(* Logix 5000 project; controller NorthLineDepalletizerPLC vendor 1 type 14 code 106 rev 33.11; software revision 33.00; part 3 of 4 *)
(* tags used below, declared in another part *)
   AcknowledgeHeightCheck : ALIAS FOR YRC1000_Rbt_Ctlr:O.Data[4].4;
   AcknowledgeLevelCheck : ALIAS FOR YRC1000_Rbt_Ctlr:O.Data[6].4;
   AcknowledgePalletTooTall : ALIAS FOR YRC1000_Rbt_Ctlr:O.Data[7].4;
   ActiveUserFrame : DINT;   // Currently Active Pallet
   AirPressure : ALIAS FOR YRC1000_Rbt_Ctlr:I.Data[1].4;
   Alarm : ALIAS FOR YRC1000_Rbt_Ctlr:I.Data[8].3;
   AngleHeightCheck : ALIAS FOR YRC1000_Rbt_Ctlr:I.Data[10].4;
   AtHomePosition : ALIAS FOR YRC1000_Rbt_Ctlr:I.Data[5].2;
   CameraFailed : ALIAS FOR YRC1000_Rbt_Ctlr:O.Data[5].7;
   CapacitiveSensorValue : DINT;
   CoilType : DINT;   // 1: 17" 2: 30" 3: 41"
   CompleteState : DINT;
   ConveyorApproach : YRC1000_POSITION_VAR;
   ConveyorBeforePlace : YRC1000_POSITION_VAR;
   ConveyorIn : YRC1000_POSITION_VAR;
   ConveyorOver : YRC1000_POSITION_VAR;
   Corner1Dist : DINT;
   Corner2Dist : DINT;
   Corner3Dist : DINT;
   Corner4Dist : DINT;
   Cos30 : REAL;
   Cos45 : REAL;
   CurrentPos : REAL[6];   // Current position of the active TCP on the robot
   CurrentPosition_micro : YRC1000_POSITION_VAR;
   delay_ActiveUserFrame : TIMER;
   delay_CurrentPos : TIMER;
   delay_Read_PartCount : TIMER;
   delay_Read_RobotCurrentTask : TIMER;
   DiffHeightCheckVal : DINT;   // Difference between the highest and shortest corners of a pallet
   DistanceSensorValue_micro : DINT;
   DoorRequestAccess : ALIAS FOR YRC1000_Rbt_Ctlr:I.Data[1].0;
   DoorUnlocked : ALIAS FOR YRC1000_Rbt_Ctlr:I.Data[1].7;
   err_CameraFailed : BOOL;
   err_HeightCheckInconsistent : ALIAS FOR YRC1000_Rbt_Ctlr:O.Data[6].3;
   err_RobotPickupFailed : ALIAS FOR YRC1000_Rbt_Ctlr:I.Data[10].3;
   ExternalHold : ALIAS FOR YRC1000_Rbt_Ctlr:O.Data[0].1;
   Gripper_Extended : ALIAS FOR YRC1000_Rbt_Ctlr:O.Data[5].0;
   Gripper_HoldingPart : ALIAS FOR YRC1000_Rbt_Ctlr:O.Data[4].7;
   Gripper_Retracted : ALIAS FOR YRC1000_Rbt_Ctlr:O.Data[5].1;
   HeightCheck1 : ALIAS FOR YRC1000_Rbt_Ctlr:I.Data[9].0;
   HeightCheck2 : ALIAS FOR YRC1000_Rbt_Ctlr:I.Data[9].1;
   HeightCheck3 : ALIAS FOR YRC1000_Rbt_Ctlr:I.Data[9].2;
   HeightCheck4 : ALIAS FOR YRC1000_Rbt_Ctlr:I.Data[9].3;
   HeightCheckAngled : REAL;
   HeightCheckAvg : DINT;
   HeightCheckTotal : DINT;
   HighestCorner : DINT;   // Index of the highest corner on a quad-stack pallet
   i : DINT;
   IFM_Device_Disconnected : BOOL;
   InHomePosition : ALIAS FOR YRC1000_Rbt_Ctlr:O.Data[5].6;
   InRemote : ALIAS FOR YRC1000_Rbt_Ctlr:I.Data[8].5;
   j : DINT;
   JobResults : PatternResult[4];   // Organized results from the most recent camera image
   LeftConveyorPresent : ALIAS FOR YRC1000_Rbt_Ctlr:O.Data[7].6;
   LeftEdgeFound : ALIAS FOR YRC1000_Rbt_Ctlr:O.Data[6].7;
   LeftPalletComplete : ALIAS FOR YRC1000_Rbt_Ctlr:O.Data[4].0;
   LeftPalletPresent : ALIAS FOR YRC1000_Rbt_Ctlr:O.Data[7].1;
   LevelCheck1 : ALIAS FOR YRC1000_Rbt_Ctlr:I.Data[10].7;
   LevelCheck2 : ALIAS FOR YRC1000_Rbt_Ctlr:I.Data[11].0;
   LevelCheck3 : ALIAS FOR YRC1000_Rbt_Ctlr:I.Data[11].1;
   LevelCheckBad : ALIAS FOR YRC1000_Rbt_Ctlr:O.Data[7].3;
   LevelCheckDone : ALIAS FOR YRC1000_Rbt_Ctlr:O.Data[6].5;
   LevelCheckStopPoint : DINT;
   LoopsFound : BOOL;   // Used to determine if we are looking at the wrong end of a single-stack coil
   MaxHeightCheckVal : DINT;
   MinHeightCheckVal : DINT;
   msg_Read_ActiveUserFrame : MESSAGE;
   msg_Read_CurrentPosition : MESSAGE;
   msg_Read_CurrentRobotTask : MESSAGE;
   msg_Read_PartCount : MESSAGE;
   msg_Read_SearchLocation : MESSAGE;
   msg_Write_ActiveUserFrame : MESSAGE;
   msg_Write_CoilLocation : MESSAGE;
   msg_Write_CoilType : MESSAGE;
   msg_Write_ConveyorApproach : MESSAGE;
   msg_Write_ConveyorBeforePlace : MESSAGE;
   msg_Write_ConveyorIn : MESSAGE;
   msg_Write_ConveyorOver : MESSAGE;
   msg_Write_HeightCheckAverage : MESSAGE;
   msg_Write_HighestCorner : MESSAGE;
   msg_Write_PartCount : MESSAGE;
   msg_Write_SearchLocation : MESSAGE;
   ons_IncPickFailCount : BOOL;
   ons_Reset_PC_HeightCheck : BOOL;
   ons_StartHeightCheck : BOOL;
   ons_StartLevelCheck : BOOL;
   p : DINT;
   PalletTooTall : ALIAS FOR YRC1000_Rbt_Ctlr:I.Data[9].6;
   PartCount : DINT;   // Number of coils the robot has placed on either conveyor
   PartID : DINT;
   PartLength_Current : DINT;   // 17" = 432 mm 30" = 762 mm 41" = 1041 mm
   PartRows_Current : DINT;
   PartThickness_Current : REAL;   // 2r = 34.1 - 34.8 mm 3r = 51.1 - 51.8 mm 4r = 68.2 - 68.9 mm
   PartWidth_Current : DINT;   // 14" = 356 mm 16" = 406 mm 20" = 508 mm 22" = 559 mm 24" = 610 mm 28" = 711 mm 32" = 813 mm
   PickFailCount : COUNTER;
   PickFailedThreeTimes : ALIAS FOR YRC1000_Rbt_Ctlr:O.Data[7].5;
   PickupErrorAcknowledge : ALIAS FOR YRC1000_Rbt_Ctlr:O.Data[5].5;
   QuadStack : ALIAS FOR YRC1000_Rbt_Ctlr:O.Data[4].3;
   Queue_PartCount : DINT[4];   // Queue of Part Counts to help keep track of what part info the Fanuc needs
   Queue_PartID : DINT[4];   // Queue of Part IDs to send to the Fanuc
   Queue_PartLength : DINT[4];   // Queue of Part Lengths to send to the Fanuc
   Queue_PartWidth : DINT[4];   // Queue of Part Widths to send to the Fanuc
   Read_ActiveUserFrame : BOOL;
   Read_CurrentPosition : BOOL;
   Read_CurrentRobotTask : BOOL;
   Read_PartCount : BOOL;
   Read_SearchLocation : BOOL;
   recovery_CameraFailed : BOOL;
   recovery_HeightCheckFailed : BOOL;
   recovery_PalletTooTall : BOOL;
   recovery_PickupFailed : BOOL;
   Reset : ALIAS FOR YRC1000_Rbt_Ctlr:I.Data[1].1;
   RightConveyorPresent : ALIAS FOR YRC1000_Rbt_Ctlr:O.Data[7].7;
   RightEdgeFound : ALIAS FOR YRC1000_Rbt_Ctlr:O.Data[7].0;
   RightPalletComplete : ALIAS FOR YRC1000_Rbt_Ctlr:O.Data[4].1;
   RightPalletPresent : ALIAS FOR YRC1000_Rbt_Ctlr:O.Data[7].2;
   RobotCurrentPalletComplete : ALIAS FOR YRC1000_Rbt_Ctlr:I.Data[10].6;
   RobotExternalEStop : ALIAS FOR YRC1000_Rbt_Ctlr:I.Data[4].1;
   RobotTeachPendantEStop : ALIAS FOR YRC1000_Rbt_Ctlr:I.Data[4].2;
   Running : ALIAS FOR YRC1000_Rbt_Ctlr:I.Data[8].0;
   RunPalletComplete : BOOL;
   SafetyCircuitBroken : ALIAS FOR YRC1000_Rbt_Ctlr:I.Data[4].0;
   SelectedJobID : DINT;
   SingleStack : ALIAS FOR YRC1000_Rbt_Ctlr:O.Data[4].2;
   StackLight_Blue : ALIAS FOR YRC1000_Rbt_Ctlr:O.Data[1].3;
   StackLight_Green : ALIAS FOR YRC1000_Rbt_Ctlr:O.Data[1].5;
   StackLight_Red : ALIAS FOR YRC1000_Rbt_Ctlr:O.Data[1].2;
   StackLight_White : ALIAS FOR YRC1000_Rbt_Ctlr:O.Data[1].1;
   StackLight_Yellow : ALIAS FOR YRC1000_Rbt_Ctlr:O.Data[1].4;
   state_HeightCheck : DINT;
   state_LevelCheck : DINT;
   state_PalletComplete : DINT;
   timer_HoldingPart : TIMER;
   ToPC_ActivePallet : DINT;
   ToPC_AirPressure : DINT;
   ToPC_CameraFailed : DINT;
   ToPC_CellStatus : DINT;
   ToPC_DoorStatus : DINT;
   ToPC_HeightCheckFailed : DINT;
   ToPC_InRemote : DINT;
   ToPC_LeftConveyorSensor : DINT;
   ToPC_LeftPalletStatus : DINT;
   ToPC_PalletTooTall : DINT;
   ToPC_PickupFailed : DINT;
   ToPC_RightConveyorSensor : DINT;
   ToPC_RightPalletStatus : DINT;
   ToPC_RobotAlarm : DINT;
   ToPC_RobotEStop : DINT;
   ToPC_RobotRunning : DINT;
   ToPC_RobotSafetyStop : DINT;
   ToPC_ToolStatus : DINT;
   Write_ActiveUserFrame : BOOL;
   write_ActiveUserFrame_L : BOOL;
   Write_ActiveUserFrame_R : BOOL;
   Write_CoilLocation : BOOL;
   Write_CoilType : BOOL;
   Write_ConveyorPositions : BOOL;
   Write_HeightCheckAverage : BOOL;
   write_HighestCorner : BOOL;
   Write_PartCount : BOOL;
   Write_SearchLocation : BOOL;
(* MainProgram, continued *)

ROUTINE PC_TagVariables   (* ladder *)
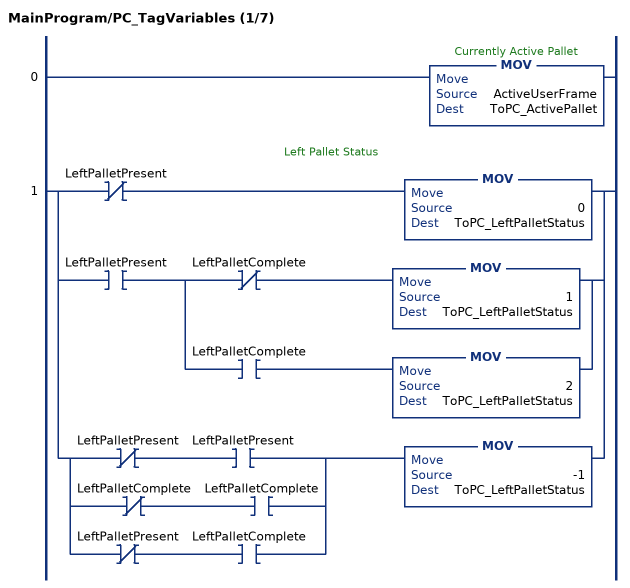
   0: MOV(ActiveUserFrame,ToPC_ActivePallet);
   // Left Pallet Status
   1: [XIO(LeftPalletPresent) MOV(0,ToPC_LeftPalletStatus) ,XIC(LeftPalletPresent) [XIO(LeftPalletComplete) MOV(1,ToPC_LeftPalletStatus) ,XIC(LeftPalletComplete) MOV(2,ToPC_LeftPalletStatus) ] ,[XIO(LeftPalletPresent) XIC(LeftPalletPresent) ,XIO(LeftPalletComplete) XIC(LeftPalletComplete) ,XIO(LeftPalletPresent) XIC(LeftPalletComplete) ] MOV(-1,ToPC_LeftPalletStatus) ];
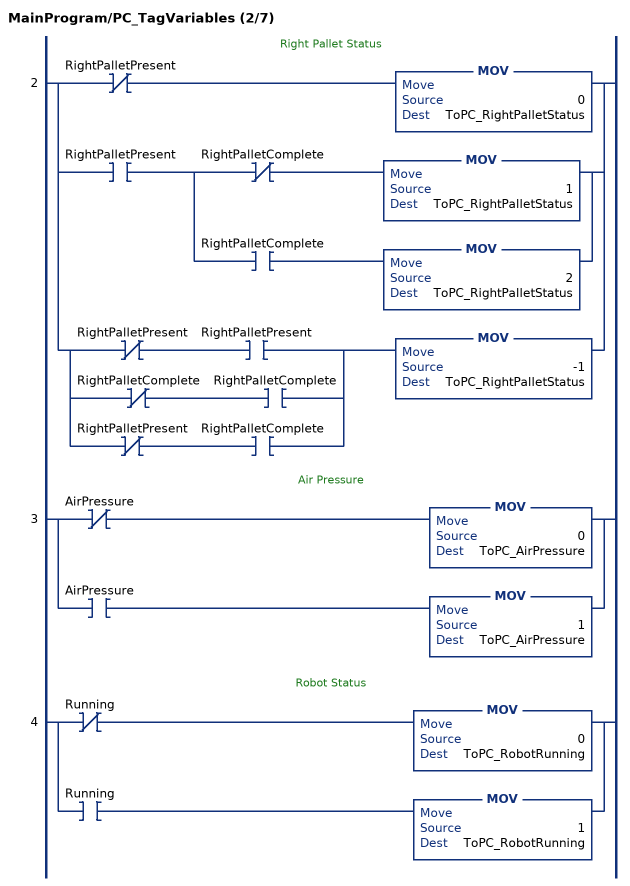
   // Right Pallet Status
   2: [XIO(RightPalletPresent) MOV(0,ToPC_RightPalletStatus) ,XIC(RightPalletPresent) [XIO(RightPalletComplete) MOV(1,ToPC_RightPalletStatus) ,XIC(RightPalletComplete) MOV(2,ToPC_RightPalletStatus) ] ,[XIO(RightPalletPresent) XIC(RightPalletPresent) ,XIO(RightPalletComplete) XIC(RightPalletComplete) ,XIO(RightPalletPresent) XIC(RightPalletComplete) ] MOV(-1,ToPC_RightPalletStatus) ];
   // Air Pressure
   3: [XIO(AirPressure) MOV(0,ToPC_AirPressure) ,XIC(AirPressure) MOV(1,ToPC_AirPressure) ];
   // Robot Status
   4: [XIO(Running) MOV(0,ToPC_RobotRunning) ,XIC(Running) MOV(1,ToPC_RobotRunning) ];
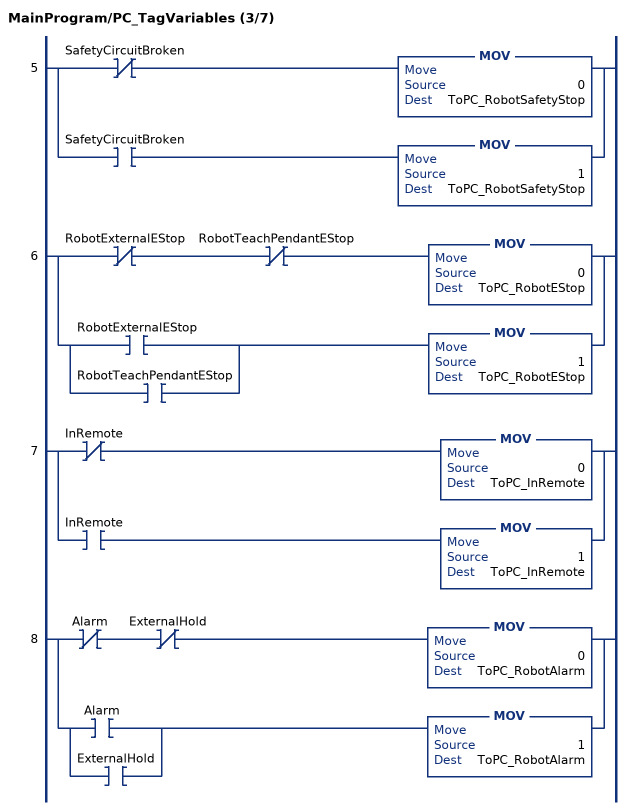
   5: [XIO(SafetyCircuitBroken) MOV(0,ToPC_RobotSafetyStop) ,XIC(SafetyCircuitBroken) MOV(1,ToPC_RobotSafetyStop) ];
   6: [XIO(RobotExternalEStop) XIO(RobotTeachPendantEStop) MOV(0,ToPC_RobotEStop) ,[XIC(RobotExternalEStop) ,XIC(RobotTeachPendantEStop) ] MOV(1,ToPC_RobotEStop) ];
   7: [XIO(InRemote) MOV(0,ToPC_InRemote) ,XIC(InRemote) MOV(1,ToPC_InRemote) ];
   8: [XIO(Alarm) XIO(ExternalHold) MOV(0,ToPC_RobotAlarm) ,[XIC(Alarm) ,XIC(ExternalHold) ] MOV(1,ToPC_RobotAlarm) ];
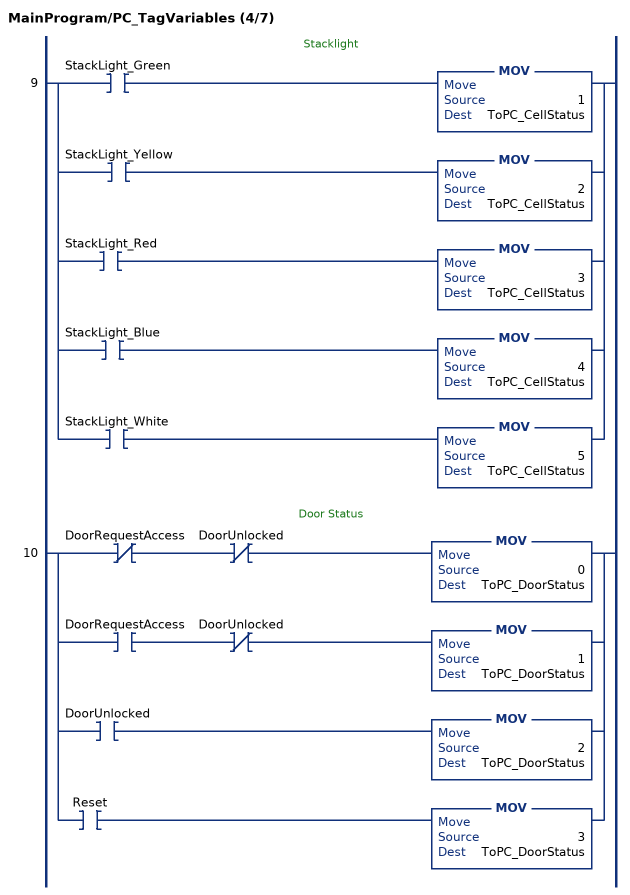
   // Stacklight
   9: [XIC(StackLight_Green) MOV(1,ToPC_CellStatus) ,XIC(StackLight_Yellow) MOV(2,ToPC_CellStatus) ,XIC(StackLight_Red) MOV(3,ToPC_CellStatus) ,XIC(StackLight_Blue) MOV(4,ToPC_CellStatus) ,XIC(StackLight_White) MOV(5,ToPC_CellStatus) ];
   // Door Status
   10: [XIO(DoorRequestAccess) XIO(DoorUnlocked) MOV(0,ToPC_DoorStatus) ,XIC(DoorRequestAccess) XIO(DoorUnlocked) MOV(1,ToPC_DoorStatus) ,XIC(DoorUnlocked) MOV(2,ToPC_DoorStatus) ,XIC(Reset) MOV(3,ToPC_DoorStatus) ];
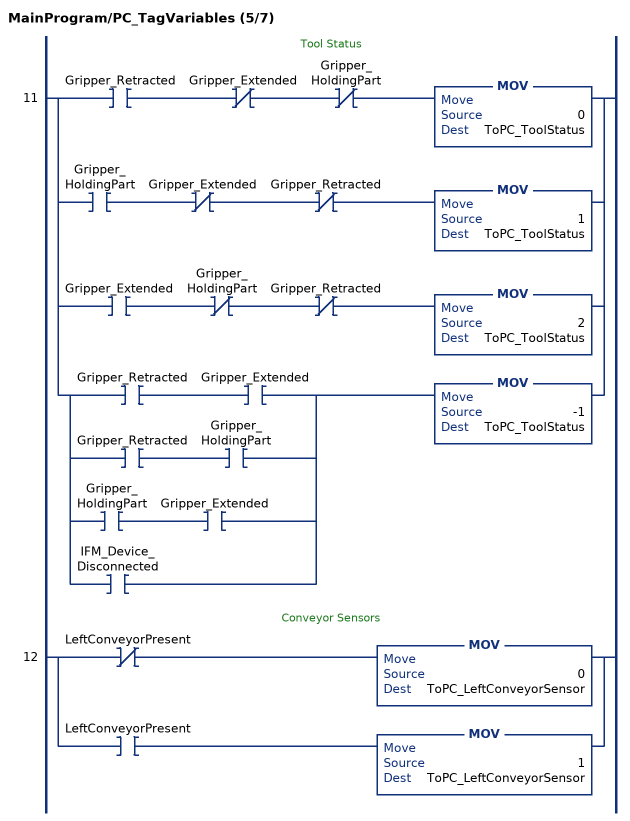
   // Tool Status
   11: [XIC(Gripper_Retracted) XIO(Gripper_Extended) XIO(Gripper_HoldingPart) MOV(0,ToPC_ToolStatus) ,XIC(Gripper_HoldingPart) XIO(Gripper_Extended) XIO(Gripper_Retracted) MOV(1,ToPC_ToolStatus) ,XIC(Gripper_Extended) XIO(Gripper_HoldingPart) XIO(Gripper_Retracted) MOV(2,ToPC_ToolStatus) ,[XIC(Gripper_Retracted) XIC(Gripper_Extended) ,XIC(Gripper_Retracted) XIC(Gripper_HoldingPart) ,XIC(Gripper_HoldingPart) XIC(Gripper_Extended) ,XIC(IFM_Device_Disconnected) ] MOV(-1,ToPC_ToolStatus) ];
   // Conveyor Sensors
   12: [XIO(LeftConveyorPresent) MOV(0,ToPC_LeftConveyorSensor) ,XIC(LeftConveyorPresent) MOV(1,ToPC_LeftConveyorSensor) ];
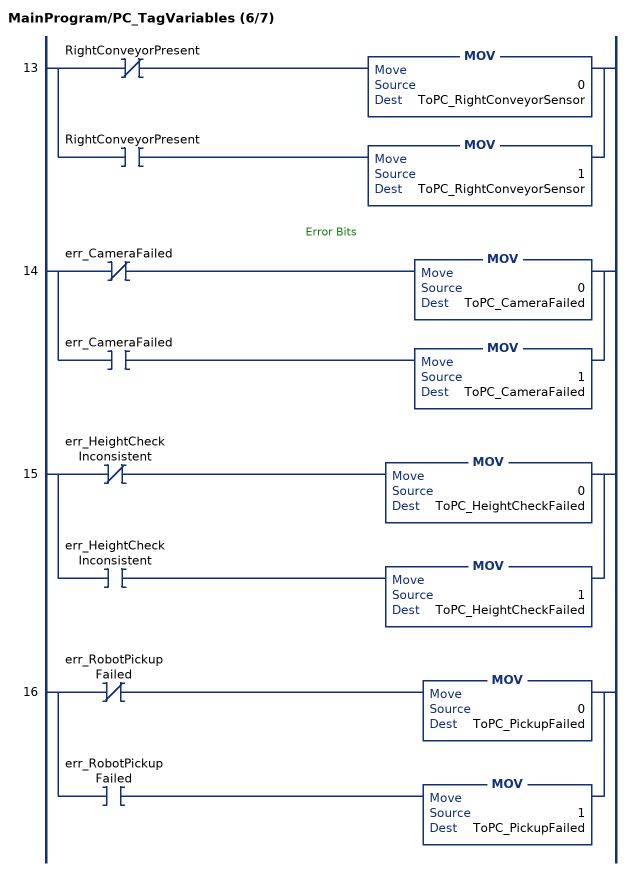
   13: [XIO(RightConveyorPresent) MOV(0,ToPC_RightConveyorSensor) ,XIC(RightConveyorPresent) MOV(1,ToPC_RightConveyorSensor) ];
   // Error Bits
   14: [XIO(err_CameraFailed) MOV(0,ToPC_CameraFailed) ,XIC(err_CameraFailed) MOV(1,ToPC_CameraFailed) ];
   15: [XIO(err_HeightCheckInconsistent) MOV(0,ToPC_HeightCheckFailed) ,XIC(err_HeightCheckInconsistent) MOV(1,ToPC_HeightCheckFailed) ];
   16: [XIO(err_RobotPickupFailed) MOV(0,ToPC_PickupFailed) ,XIC(err_RobotPickupFailed) MOV(1,ToPC_PickupFailed) ];
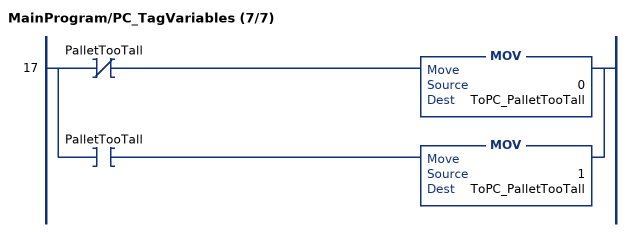
   17: [XIO(PalletTooTall) MOV(0,ToPC_PalletTooTall) ,XIC(PalletTooTall) MOV(1,ToPC_PalletTooTall) ];
END_ROUTINE

ROUTINE SaveImageResults   (* structured text *)
   /*
   	Simple loop going through all the information given by the camera after capturing an image
   	Loop through the 28 possible patterns
   	Each pattern has 4 parts: Angle, Score, X, and Y
   */
   
   for i := 0 to 2 by 1 do
   	j := i * 4;
   	JobResults[i].Angle := cam:I.InspectionResults[j];
   	JobResults[i].Score := cam:I.InspectionResults[j + 1];
   	JobResults[i].X := cam:I.InspectionResults[j + 2];
   	JobResults[i].Y := cam:I.InspectionResults[j + 3];
   end_for;
   
   if SelectedJobID = 2832 then
   	if cam:I.InspectionResults[12] > 0 then
   		LoopsFound := 1;
   	else
   		LoopsFound := 0;
   	end_if;
   end_if;
   
   if SelectedJobID = 3041 then
   	if cam:I.InspectionResults[12] > 0 then
   		LeftEdgeFound := 1;
   	else
   		LeftEdgeFound := 0;
   	end_if;
   	if cam:I.InspectionResults[13] > 0 then
   		RightEdgeFound := 1;
   	else
   		RightEdgeFound := 0;
   	end_if;
   	if cam:I.InspectionResults[14] > 0 then
   		LoopsFound := 1;
   	else
   		LoopsFound := 0;
   	end_if;
   end_if;
END_ROUTINE
END_PROGRAM

PROGRAM Motoman   (* main routine Main *)

ROUTINE AddPartToQueue   (* structured text *)
   // Determine unique Part ID that can be sent to the Fanuc
   if PartLength_Current = 432 then
   	if PartWidth_Current = 356 then
   		PartID := 1;
   	elsif PartWidth_Current = 406 then
   		PartID := 2;
   	elsif PartWidth_Current = 508 then
   		if PartRows_Current = 2 then
   			PartID := 3;
   		elsif PartRows_Current = 3 then
   			PartID := 4;
   		end_if;
   	elsif PartWidth_Current = 559 then
   		PartID := 5;
   	elsif PartWidth_Current = 610 then
   		PartID := 6;
   	elsif PartWidth_Current = 711 then
   		if PartRows_Current = 3 then
   			PartID := 7;
   		elsif PartRows_Current = 4 then
   			PartID := 8;
   		end_if;
   	elsif PartWidth_Current = 813 then
   		PartID := 9;
   	end_if;
   elsif PartLength_Current = 762 then
   	if PartRows_Current = 2 then
   		PartID := 10;
   	elsif PartRows_Current = 3 then
   		PartID := 11;
   	end_if;
   elsif PartLength_Current = 1041 then
   	if PartRows_Current = 3 then
   		PartID := 12;
   	elsif PartRows_Current = 4 then
   		PartID := 13;
   	end_if;
   end_if;
   
   // Add information about the new part to a bunch of arrays
   for p := 1 to 3 do
   	if Queue_PartID[p] = 0 then
   		Queue_PartCount[p-1] := PartCount;
   		Queue_PartID[p] := PartID;
   		Queue_PartLength[p] := PartLength_Current;
   		Queue_PartWidth[p] := PartWidth_Current;
   
   		RET();
   	end_if;
   end_for;
   
END_ROUTINE

ROUTINE CheckForHeightOutliers   (* structured text *)
   MinHeightCheckVal := 0;
   MaxHeightCheckVal := 0;
   DiffHeightCheckVal := 0;
   
   if Corner1Dist <= Corner2Dist AND Corner1Dist <= Corner3Dist AND Corner1Dist <= Corner4Dist then
   	MinHeightCheckVal := Corner1Dist;
   	HighestCorner := 1;
   elsif Corner2Dist <= Corner1Dist AND Corner2Dist <= Corner3Dist AND Corner2Dist <= Corner4Dist then
   	MinHeightCheckVal := Corner2Dist;
   	HighestCorner := 2;
   elsif Corner3Dist <= Corner1Dist AND Corner3Dist <= Corner2Dist AND Corner3Dist <= Corner4Dist then
   	MinHeightCheckVal := Corner3Dist;
   	HighestCorner := 3;
   elsif Corner4Dist <= Corner1Dist AND Corner4Dist <= Corner2Dist AND Corner4Dist <= Corner3Dist then
   	MinHeightCheckVal := Corner4Dist;
   	HighestCorner := 4;
   end_if;
   
   if Corner1Dist >= Corner2Dist AND Corner1Dist >= Corner3Dist AND Corner1Dist >= Corner4Dist then
   	MaxHeightCheckVal := Corner1Dist;
   elsif Corner2Dist >= Corner1Dist AND Corner2Dist >= Corner3Dist AND Corner2Dist >= Corner4Dist then
   	MaxHeightCheckVal := Corner2Dist;
   elsif Corner3Dist >= Corner1Dist AND Corner3Dist >= Corner2Dist AND Corner3Dist >= Corner4Dist then
   	MaxHeightCheckVal := Corner3Dist;
   elsif Corner4Dist >= Corner1Dist AND Corner4Dist >= Corner2Dist AND Corner4Dist >= Corner3Dist then
   	MaxHeightCheckVal := Corner4Dist;
   end_if;
   
   DiffHeightCheckVal := MaxHeightCheckVal - MinHeightCheckVal;
   if DiffHeightCheckVal > 25000 AND MinHeightCheckVal < 1990000 then
   	err_HeightCheckInconsistent := 1;
   else
   	err_HeightCheckInconsistent := 0;
   end_if;
END_ROUTINE

ROUTINE ConveyorVariableData   (* structured text *)
   /*
   	The only major values that change are
   		Tool_Num depending on the Part Length and
   		Axis3_Data depending on the Part Thickness
   */
   
   // Tool Number
   if PartLength_Current = 432 then
   	ConveyorApproach.Tool_Num := 8;
   	ConveyorOver.Tool_Num := 8;
   	ConveyorIn.Tool_Num := 8;
   	ConveyorBeforePlace.Tool_Num := 8;
   	ConveyorOver.Axis5_Data := 100000;
   	ConveyorIn.Axis5_Data := 100000;
   	ConveyorBeforePlace.Axis5_Data := 100000;
   elsif PartLength_Current = 762 then
   	ConveyorApproach.Tool_Num := 9;
   	ConveyorOver.Tool_Num := 9;
   	ConveyorIn.Tool_Num := 9;
   	ConveyorBeforePlace.Tool_Num := 9;
   	ConveyorOver.Axis5_Data := 100000;
   	ConveyorIn.Axis5_Data := 100000;
   	ConveyorBeforePlace.Axis5_Data :=100000;
   elsif PartLength_Current = 1041 then
   	ConveyorApproach.Tool_Num := 10;
   	ConveyorOver.Tool_Num := 10;
   	ConveyorIn.Tool_Num := 10;
   	ConveyorBeforePlace.Tool_Num := 10;
   	ConveyorOver.Axis5_Data := 80000;
   	ConveyorIn.Axis5_Data := 80000;
   	ConveyorBeforePlace.Axis5_Data := 80000;
   end_if;
   
   // Conveyor Above Z value is dependent on Part Thickness
   ConveyorApproach.Axis3_Data := (PartThickness_Current + 100) * 1000;
   ConveyorOver.Axis3_Data := (PartThickness_Current + 100) * 1000;
   ConveyorIn.Axis3_Data := (PartThickness_Current + 5) * 1000;
   ConveyorBeforePlace.Axis3_Data := (PartThickness_Current + 5) * 1000;
END_ROUTINE

ROUTINE ErrorBits   (* ladder *)
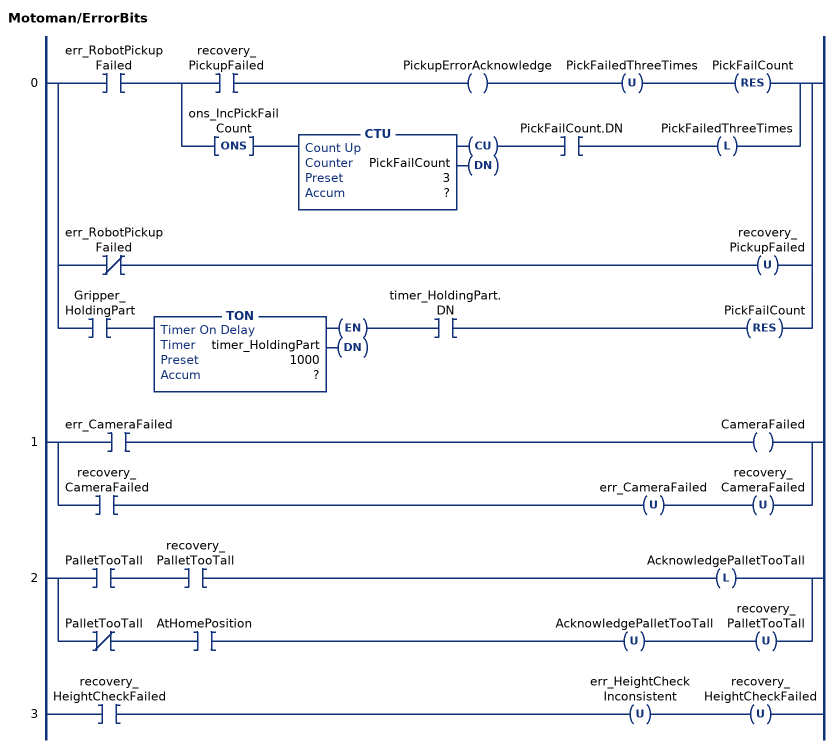
   0: [XIC(err_RobotPickupFailed) [XIC(recovery_PickupFailed) OTE(PickupErrorAcknowledge) OTU(PickFailedThreeTimes) RES(PickFailCount) ,ONS(ons_IncPickFailCount) CTU(PickFailCount,?,?) XIC(PickFailCount.DN) OTL(PickFailedThreeTimes) ] ,XIO(err_RobotPickupFailed) OTU(recovery_PickupFailed) ,XIC(Gripper_HoldingPart) TON(timer_HoldingPart,?,?) XIC(timer_HoldingPart.DN) RES(PickFailCount) ];
   1: [XIC(err_CameraFailed) OTE(CameraFailed) ,XIC(recovery_CameraFailed) OTU(err_CameraFailed) OTU(recovery_CameraFailed) ];
   2: [XIC(PalletTooTall) XIC(recovery_PalletTooTall) OTL(AcknowledgePalletTooTall) ,XIO(PalletTooTall) XIC(AtHomePosition) OTU(AcknowledgePalletTooTall) OTU(recovery_PalletTooTall) ];
   3: XIC(recovery_HeightCheckFailed)OTU(err_HeightCheckInconsistent)OTU(recovery_HeightCheckFailed);
END_ROUTINE

ROUTINE HeightCheck   (* ladder *)
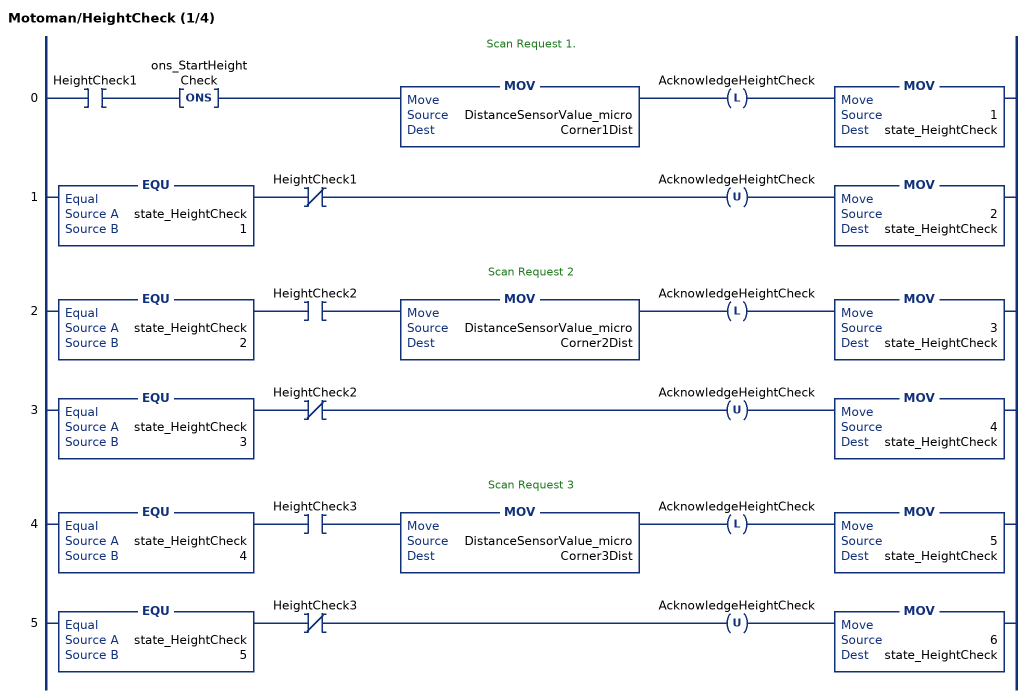
   // Scan Request 1.
   0: XIC(HeightCheck1)ONS(ons_StartHeightCheck)MOV(DistanceSensorValue_micro,Corner1Dist)OTL(AcknowledgeHeightCheck)MOV(1,state_HeightCheck);
   1: EQU(state_HeightCheck,1)XIO(HeightCheck1)OTU(AcknowledgeHeightCheck)MOV(2,state_HeightCheck);
   // Scan Request 2
   2: EQU(state_HeightCheck,2)XIC(HeightCheck2)MOV(DistanceSensorValue_micro,Corner2Dist)OTL(AcknowledgeHeightCheck)MOV(3,state_HeightCheck);
   3: EQU(state_HeightCheck,3)XIO(HeightCheck2)OTU(AcknowledgeHeightCheck)MOV(4,state_HeightCheck);
   // Scan Request 3
   4: EQU(state_HeightCheck,4)XIC(HeightCheck3)MOV(DistanceSensorValue_micro,Corner3Dist)OTL(AcknowledgeHeightCheck)MOV(5,state_HeightCheck);
   5: EQU(state_HeightCheck,5)XIO(HeightCheck3)OTU(AcknowledgeHeightCheck)MOV(6,state_HeightCheck);
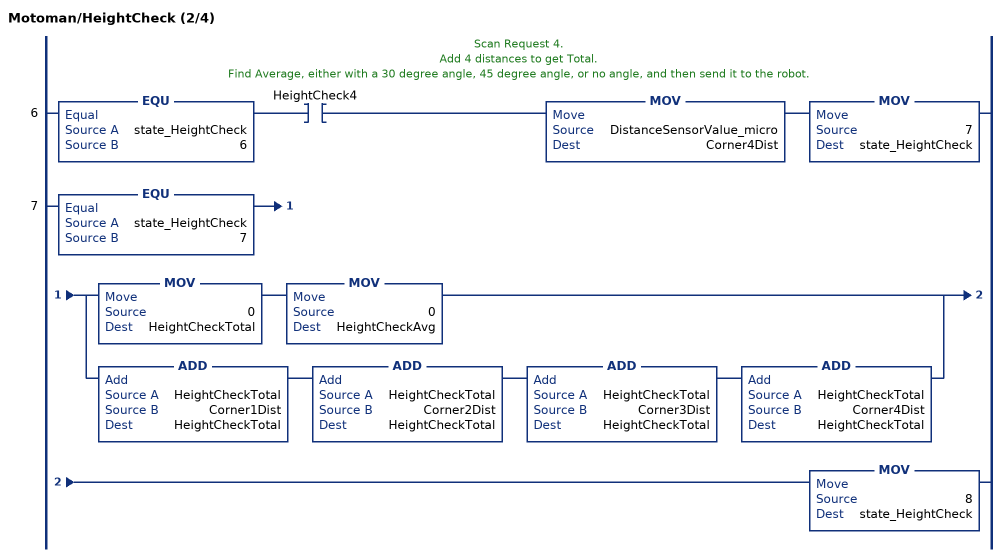
   // Scan Request 4.
   // Add 4 distances to get Total.
   // Find Average, either with a 30 degree angle, 45 degree angle, or no angle, and then send it to the robot.
   6: EQU(state_HeightCheck,6)XIC(HeightCheck4)MOV(DistanceSensorValue_micro,Corner4Dist)MOV(7,state_HeightCheck);
   7: EQU(state_HeightCheck,7)[MOV(0,HeightCheckTotal) MOV(0,HeightCheckAvg) ,ADD(HeightCheckTotal,Corner1Dist,HeightCheckTotal) ADD(HeightCheckTotal,Corner2Dist,HeightCheckTotal) ADD(HeightCheckTotal,Corner3Dist,HeightCheckTotal) ADD(HeightCheckTotal,Corner4Dist,HeightCheckTotal) ]MOV(8,state_HeightCheck);
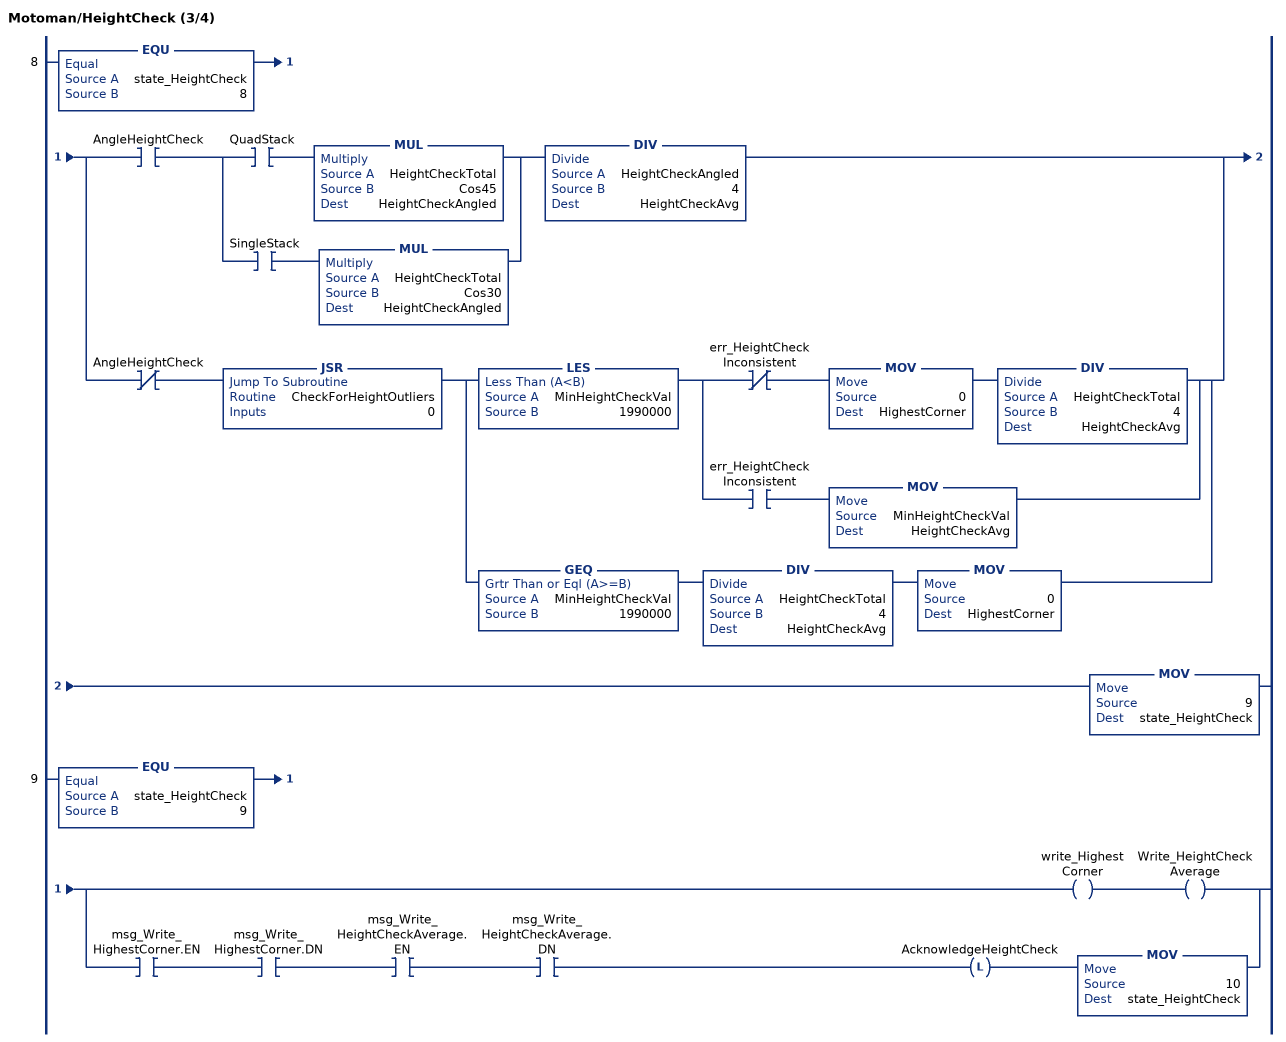
   8: EQU(state_HeightCheck,8)[XIC(AngleHeightCheck) [XIC(QuadStack) MUL(HeightCheckTotal,Cos45,HeightCheckAngled) ,XIC(SingleStack) MUL(HeightCheckTotal,Cos30,HeightCheckAngled) ] DIV(HeightCheckAngled,4,HeightCheckAvg) ,XIO(AngleHeightCheck) JSR(CheckForHeightOutliers,0) [LES(MinHeightCheckVal,1990000) [XIO(err_HeightCheckInconsistent) MOV(0,HighestCorner) DIV(HeightCheckTotal,4,HeightCheckAvg) ,XIC(err_HeightCheckInconsistent) MOV(MinHeightCheckVal,HeightCheckAvg) ] ,GEQ(MinHeightCheckVal,1990000) DIV(HeightCheckTotal,4,HeightCheckAvg) MOV(0,HighestCorner) ] ]MOV(9,state_HeightCheck);
   9: EQU(state_HeightCheck,9)[OTE(write_HighestCorner) OTE(Write_HeightCheckAverage) ,XIC(msg_Write_HighestCorner.EN) XIC(msg_Write_HighestCorner.DN) XIC(msg_Write_HeightCheckAverage.EN) XIC(msg_Write_HeightCheckAverage.DN) OTL(AcknowledgeHeightCheck) MOV(10,state_HeightCheck) ];
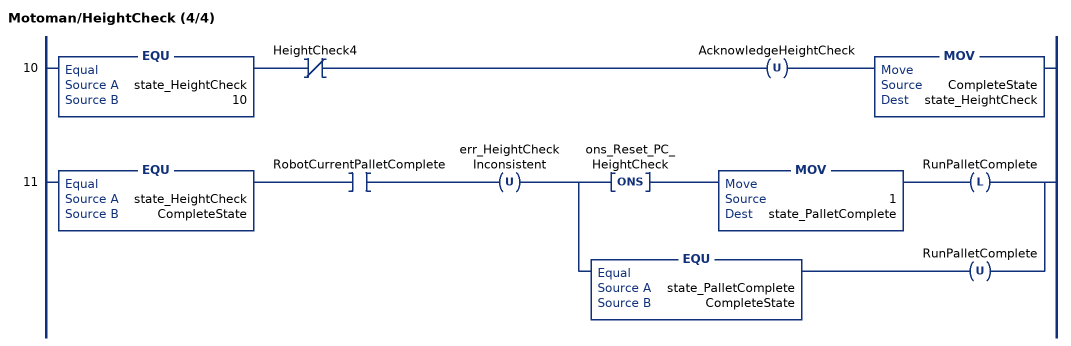
   10: EQU(state_HeightCheck,10)XIO(HeightCheck4)OTU(AcknowledgeHeightCheck)MOV(CompleteState,state_HeightCheck);
   11: EQU(state_HeightCheck,CompleteState)XIC(RobotCurrentPalletComplete)OTU(err_HeightCheckInconsistent)[ONS(ons_Reset_PC_HeightCheck) MOV(1,state_PalletComplete) OTL(RunPalletComplete) ,EQU(state_PalletComplete,CompleteState) OTU(RunPalletComplete) ];
END_ROUTINE

ROUTINE LevelCheck   (* ladder *)
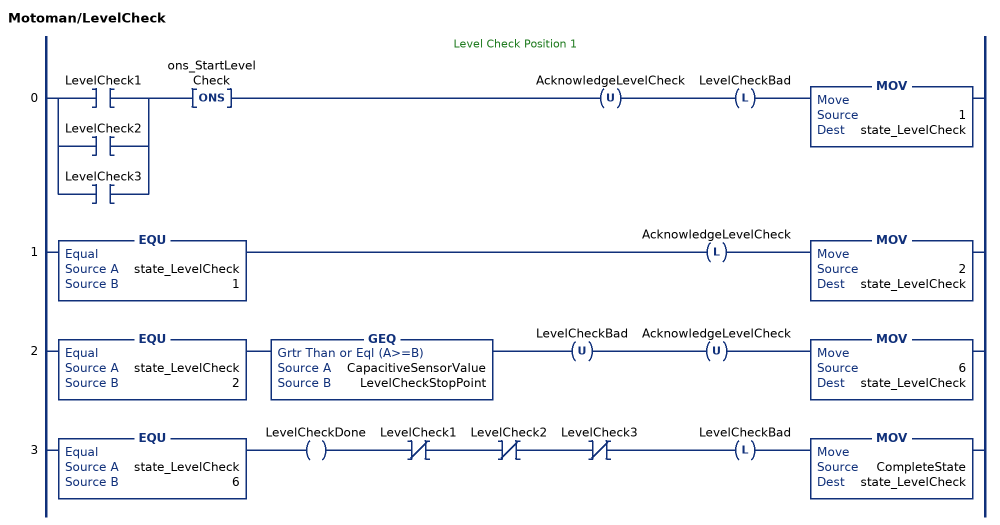
   // Level Check Position 1
   0: [XIC(LevelCheck1) ,XIC(LevelCheck2) ,XIC(LevelCheck3) ]ONS(ons_StartLevelCheck)OTU(AcknowledgeLevelCheck)OTL(LevelCheckBad)MOV(1,state_LevelCheck);
   1: EQU(state_LevelCheck,1)OTL(AcknowledgeLevelCheck)MOV(2,state_LevelCheck);
   2: EQU(state_LevelCheck,2)GEQ(CapacitiveSensorValue,LevelCheckStopPoint)OTU(LevelCheckBad)OTU(AcknowledgeLevelCheck)MOV(6,state_LevelCheck);
   3: EQU(state_LevelCheck,6)OTE(LevelCheckDone)XIO(LevelCheck1)XIO(LevelCheck2)XIO(LevelCheck3)OTL(LevelCheckBad)MOV(CompleteState,state_LevelCheck);
END_ROUTINE

ROUTINE Main   (* ladder *)
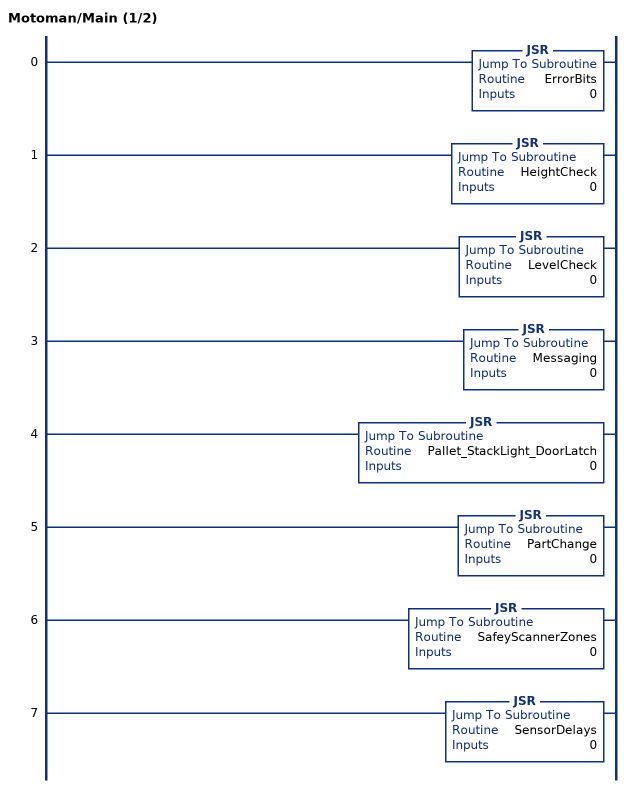
   0: JSR(ErrorBits,0);
   1: JSR(HeightCheck,0);
   2: JSR(LevelCheck,0);
   3: JSR(Messaging,0);
   4: JSR(Pallet_StackLight_DoorLatch,0);
   5: JSR(PartChange,0);
   6: JSR(SafeyScannerZones,0);
   7: JSR(SensorDelays,0);
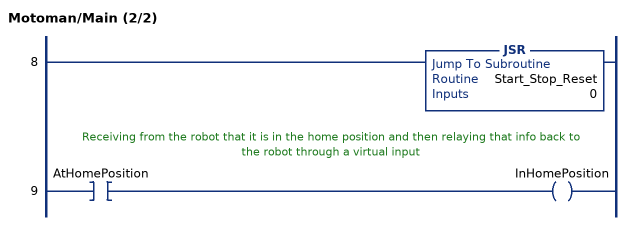
   8: JSR(Start_Stop_Reset,0);
   // Receiving from the robot that it is in the home position and then relaying that info back to the robot through a virtual input
   9: XIC(AtHomePosition)OTE(InHomePosition);
END_ROUTINE

ROUTINE Messaging   (* ladder *)
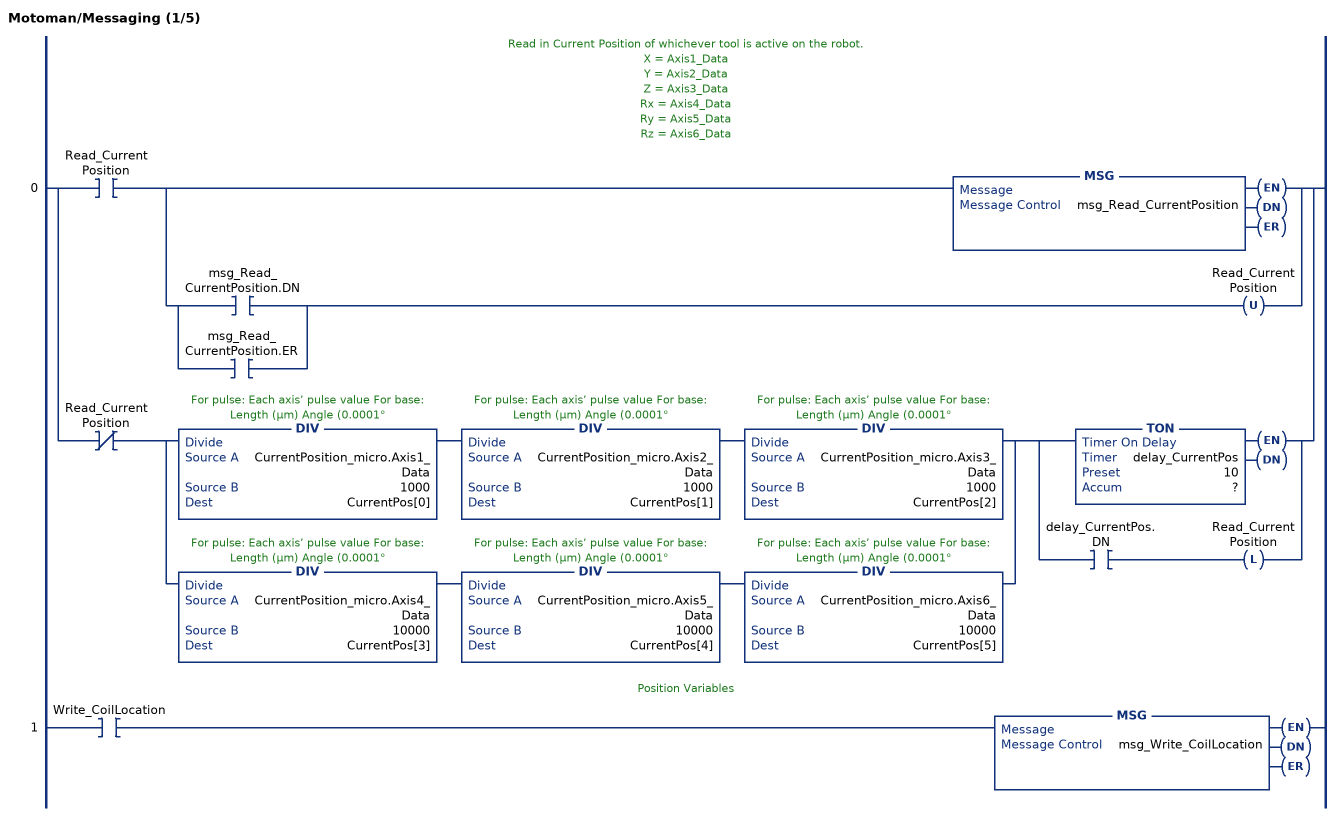
   // Read in Current Position of whichever tool is active on the robot.
   //  X = Axis1_Data
   //  Y = Axis2_Data
   //  Z = Axis3_Data
   // Rx = Axis4_Data
   // Ry = Axis5_Data
   // Rz = Axis6_Data
   0: [XIC(Read_CurrentPosition) [MSG(msg_Read_CurrentPosition) ,[XIC(msg_Read_CurrentPosition.DN) ,XIC(msg_Read_CurrentPosition.ER) ] OTU(Read_CurrentPosition) ] ,XIO(Read_CurrentPosition) [DIV(CurrentPosition_micro.Axis1_Data,1000,CurrentPos[0]) DIV(CurrentPosition_micro.Axis2_Data,1000,CurrentPos[1]) DIV(CurrentPosition_micro.Axis3_Data,1000,CurrentPos[2]) ,DIV(CurrentPosition_micro.Axis4_Data,10000,CurrentPos[3]) DIV(CurrentPosition_micro.Axis5_Data,10000,CurrentPos[4]) DIV(CurrentPosition_micro.Axis6_Data,10000,CurrentPos[5]) ] [TON(delay_CurrentPos,?,?) ,XIC(delay_CurrentPos.DN) OTL(Read_CurrentPosition) ] ];
   // Position Variables
   1: XIC(Write_CoilLocation)MSG(msg_Write_CoilLocation);
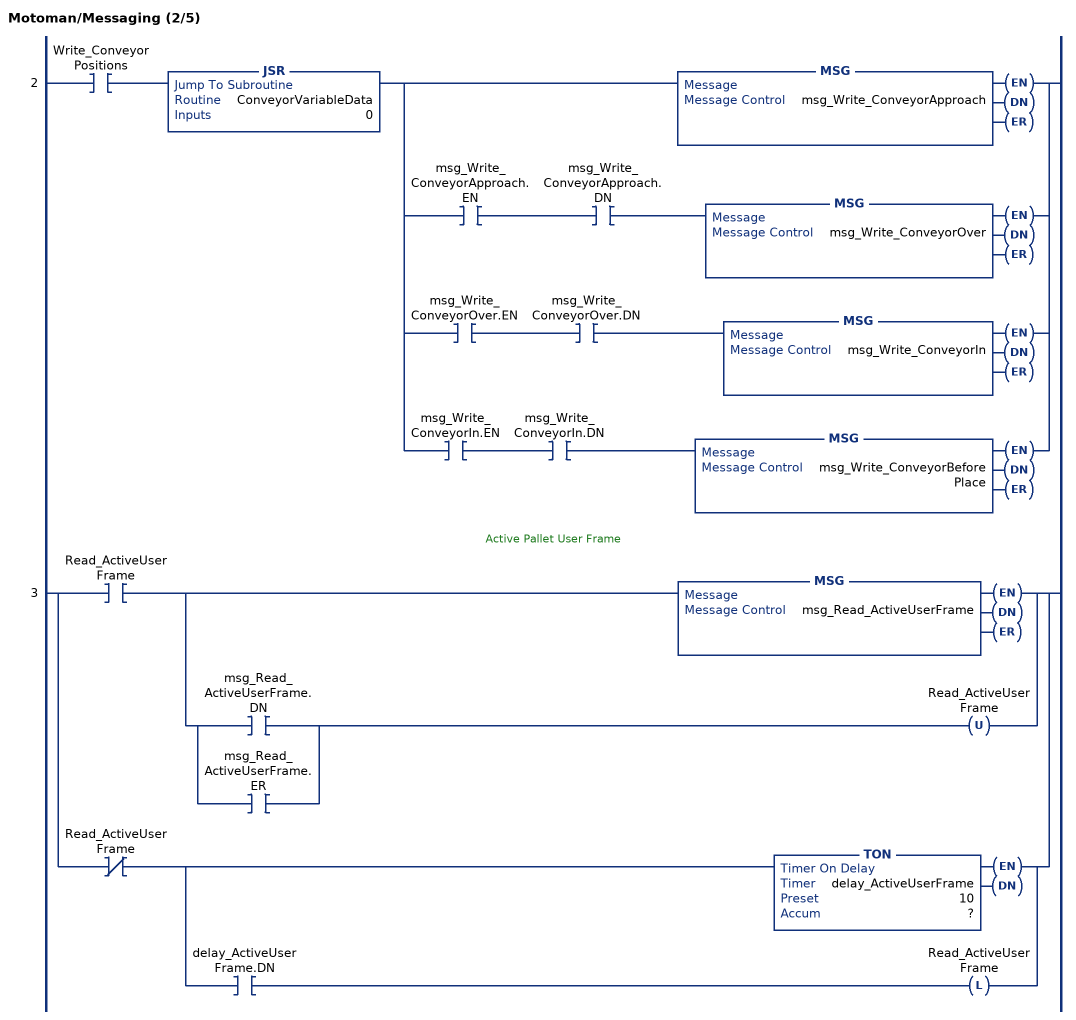
   2: XIC(Write_ConveyorPositions)JSR(ConveyorVariableData,0)[MSG(msg_Write_ConveyorApproach) ,XIC(msg_Write_ConveyorApproach.EN) XIC(msg_Write_ConveyorApproach.DN) MSG(msg_Write_ConveyorOver) ,XIC(msg_Write_ConveyorOver.EN) XIC(msg_Write_ConveyorOver.DN) MSG(msg_Write_ConveyorIn) ,XIC(msg_Write_ConveyorIn.EN) XIC(msg_Write_ConveyorIn.DN) MSG(msg_Write_ConveyorBeforePlace) ];
   // Active Pallet User Frame
   3: [XIC(Read_ActiveUserFrame) [MSG(msg_Read_ActiveUserFrame) ,[XIC(msg_Read_ActiveUserFrame.DN) ,XIC(msg_Read_ActiveUserFrame.ER) ] OTU(Read_ActiveUserFrame) ] ,XIO(Read_ActiveUserFrame) [TON(delay_ActiveUserFrame,?,?) ,XIC(delay_ActiveUserFrame.DN) OTL(Read_ActiveUserFrame) ] ];
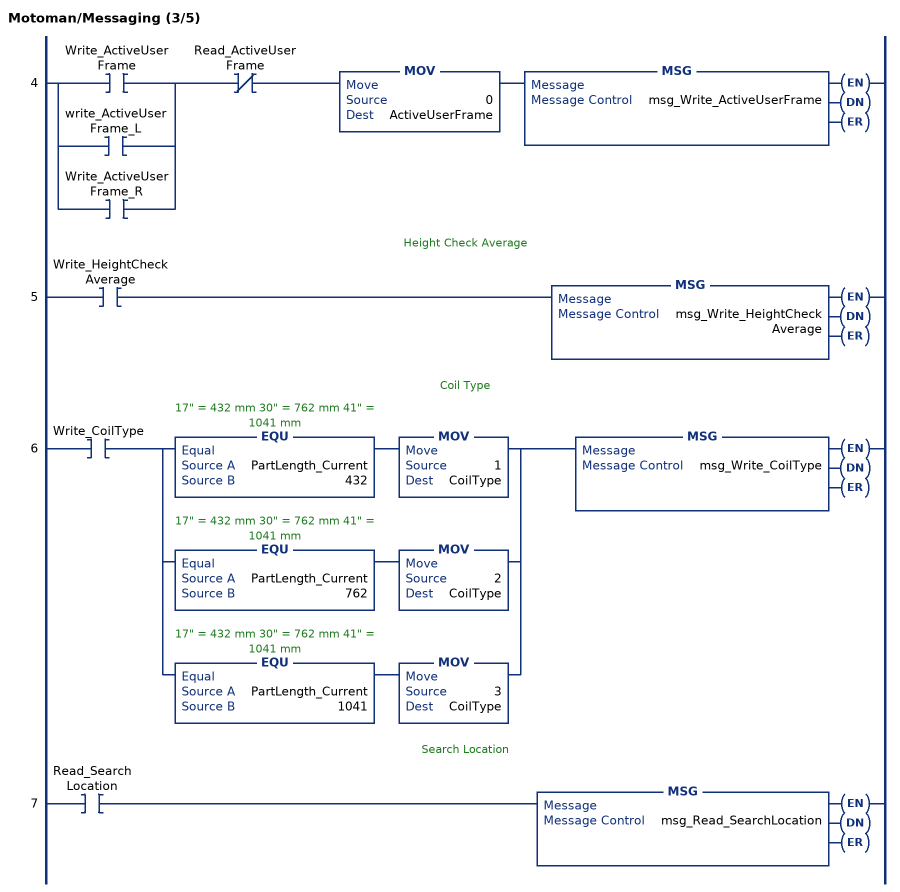
   4: [XIC(Write_ActiveUserFrame) ,XIC(write_ActiveUserFrame_L) ,XIC(Write_ActiveUserFrame_R) ]XIO(Read_ActiveUserFrame)MOV(0,ActiveUserFrame)MSG(msg_Write_ActiveUserFrame);
   // Height Check Average
   5: XIC(Write_HeightCheckAverage)MSG(msg_Write_HeightCheckAverage);
   // Coil Type
   6: XIC(Write_CoilType)[EQU(PartLength_Current,432) MOV(1,CoilType) ,EQU(PartLength_Current,762) MOV(2,CoilType) ,EQU(PartLength_Current,1041) MOV(3,CoilType) ]MSG(msg_Write_CoilType);
   // Search Location
   7: XIC(Read_SearchLocation)MSG(msg_Read_SearchLocation);
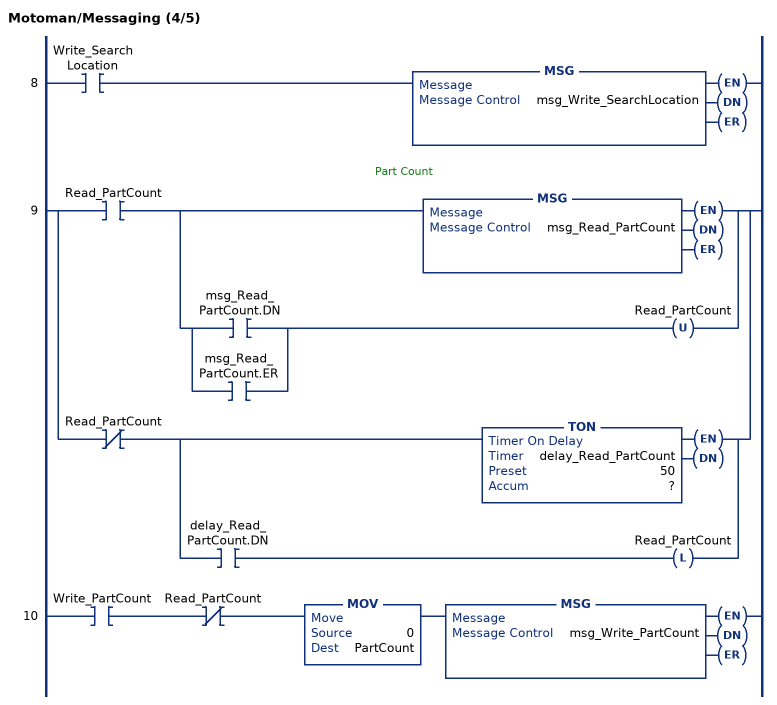
   8: XIC(Write_SearchLocation)MSG(msg_Write_SearchLocation);
   // Part Count
   9: [XIC(Read_PartCount) [MSG(msg_Read_PartCount) ,[XIC(msg_Read_PartCount.DN) ,XIC(msg_Read_PartCount.ER) ] OTU(Read_PartCount) ] ,XIO(Read_PartCount) [TON(delay_Read_PartCount,?,?) ,XIC(delay_Read_PartCount.DN) OTL(Read_PartCount) ] ];
   10: XIC(Write_PartCount)XIO(Read_PartCount)MOV(0,PartCount)MSG(msg_Write_PartCount);
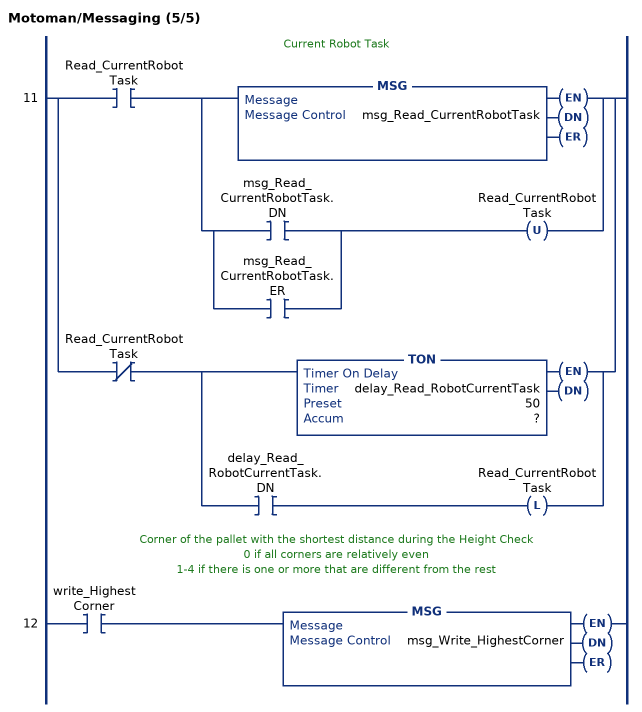
   // Current Robot Task
   11: [XIC(Read_CurrentRobotTask) [MSG(msg_Read_CurrentRobotTask) ,[XIC(msg_Read_CurrentRobotTask.DN) ,XIC(msg_Read_CurrentRobotTask.ER) ] OTU(Read_CurrentRobotTask) ] ,XIO(Read_CurrentRobotTask) [TON(delay_Read_RobotCurrentTask,?,?) ,XIC(delay_Read_RobotCurrentTask.DN) OTL(Read_CurrentRobotTask) ] ];
   // Corner of the pallet with the shortest distance during the Height Check
   //         0 if all corners are relatively even
   //         1-4 if there is one or more that are different from the rest
   12: XIC(write_HighestCorner)MSG(msg_Write_HighestCorner);
END_ROUTINE
